Staubli VAL3: resetTask.pgx

public program resetTask()
begin
  // This program kills and re-launch detection library without
  //  doing an initialization of variables.
  //
  // Input Param
  //  none       :
  //
  // Output Param
  //  none       :
  //
  //----------------------------------------------------------------
  //
  taskKill(sTASK)
  bTaskDetOK=false
  //
  taskCreate sTASK,100,detection()
  //
end
